// TIA Portal project "Conveyor_Automation_Project" (V17)

(* hardware
DEVICE "S7-1200 station_1"  S7-1200 Station
   slot 0: "Rack_0"  S7-1200 Rack  Rack  V1.0
   slot 1: "PLC_1"  CPU 1214C DC/DC/DC  6ES7 214-1AG40-0XB0  V4.5
DEVICE "HMI_1"  TP700 Comfort
   slot 0: "HMI_1"  TP700 Comfort  6AV2 124-0GC01-0AX0  17.0.0.0
   slot 1: "HMI_RT_1"  TP700 Comfort  6AV2 124-0GC01-0AX0  17.0.0.0
   slot 5: "HMI_1.IE_CP_1"  PROFINET Interface  17.0.0.0
      slot 1: "PROFINET Interface_1"  PROFINET Interface
         slot 1: "Port_1"  Port
         slot 2: "Port_2"  Port
   slot 7: "HMI_1.MPI/DP_CP_1"  MPI/DP Interface  17.0.0.0
*)

// ===== PLC "PLC_1"  CPU 1214C DC/DC/DC =====

VAR_GLOBAL   // PLC tag table "Default tag table"
   "Start_PB" AT %I0.0 : Bool;
   "Stop_PB" AT %I0.1 : Bool;
   "E_Stop" AT %I0.2 : Bool;
   "Object_Sensor" AT %I0.3 : Bool;
   "Sort_Sensor" AT %I0.4 : Bool;
   "Zone1_OL" AT %I0.5 : Bool;
   "Zone2_OL" AT %I0.6 : Bool;
   "Reset_PB" AT %I0.7 : Bool;
   "Zone1_Motor" AT %Q0.0 : Bool;
   "Zone2_Motor" AT %Q0.1 : Bool;
   "Sort_Arm" AT %Q0.2 : Bool;
   "Alarm_Light" AT %Q0.3 : Bool;
   "Run_Light" AT %Q0.4 : Bool;
   "Belt_Speed" AT %IW64 : Word;
   "VFD_Speed_Ref" AT %QW64 : Word;
END_VAR

DATA_BLOCK "Motor1_DB"   // DB1
{ S7_Optimized_Access := 'TRUE' }
VERSION : 0.1
// stored: InstanceOfName Motor_Control
"Motor_Control"
BEGIN
END_DATA_BLOCK

DATA_BLOCK "Safety_DB"   // DB2
{ S7_Optimized_Access := 'TRUE' }
VERSION : 0.1
// stored: InstanceOfName Safety logic
"Safety logic"
BEGIN
END_DATA_BLOCK

DATA_BLOCK "Motor2_DB"   // DB3
{ S7_Optimized_Access := 'TRUE' }
VERSION : 0.1
// stored: InstanceOfName Motor_Control
"Motor_Control"
BEGIN
END_DATA_BLOCK

DATA_BLOCK "Converyor_DB"   // DB4
{ S7_Optimized_Access := 'TRUE' }
VERSION : 0.1
   VAR
      System_RUnning : Bool;
      System_Fault : Bool;
      Safety_Ok : Bool;
      Auto_mode : Bool := true;
      Belt_Speed : Int;
      Belt_Speed_MS : Real;
      VFD_Output : Real;
      Speed_Setpoint : Real := 50.0;
      Good_Count : Int;
      Rject_Count : Int;
      Total_Count : Int;
      Shift_Count : Int;
      Sort_Timer : TON_TIME;
      Jam_timer : TON_TIME;
      Zone2_delay : TON_TIME;
      Good_Count_CTU : CTU_INT;
   END_VAR
   VAR RETAIN
      Reject_Count_CTU : CTU_INT;
      VFD_Output1 : Int;
   END_VAR
   VAR
      Actual_RPM : Real;
   END_VAR
BEGIN
END_DATA_BLOCK

DATA_BLOCK "Alarm_DB"   // DB5
{ S7_Optimized_Access := 'TRUE' }
VERSION : 0.1
   VAR
      Zone1_Fault : Bool;   // Zone 1 motor fault
      Zone2_Fault : Bool;   // Zone 2 motor fault
      E_Stop_Active : Bool;   // E-stop pressed
      Belt_Jam : Bool;   // Belt jam detected
      Speed_Low : Bool;   // Belt speed too low
      Any_Alarm : Bool;   // Any alarm active
      Alarm_Count : Bool;   // Total alarm count
      Alarm_Word : Word;
   END_VAR
BEGIN
END_DATA_BLOCK

DATA_BLOCK "Safety_DB_Instance"   // DB7
{ S7_Optimized_Access := 'TRUE' }
VERSION : 0.1
// stored: InstanceOfName Safety logic
"Safety logic"
BEGIN
END_DATA_BLOCK

DATA_BLOCK "Conveyor_SFC_DB"   // DB8
{ S7_Optimized_Access := 'TRUE' }
VERSION : 0.1
// stored: InstanceOfName Conveyor_SFC
"Conveyor_SFC"
BEGIN
END_DATA_BLOCK

// folder: System blocks/Program resources

DATA_BLOCK "IEC_Timer_0_DB"   // DB6
{ S7_Optimized_Access := 'TRUE' }
AUTHOR : Simatic
FAMILY : IEC
NAME : IEC_TMR
VERSION : 1.0
// stored: InstanceOfName IEC_TIMER
"IEC_TIMER"
BEGIN
END_DATA_BLOCK

// folder: (top level)

FUNCTION_BLOCK "Motor_Control"   // FB1, LAD
{ S7_Optimized_Access := 'TRUE' }
VERSION : 0.1
   VAR_INPUT
      Start : Bool;   // Start command
      Stop : Bool;   // Stop command
      Fault : Bool;   // Motor fault/overload
      Enable : Bool;   // Safety enable signal
      Auto_Mode : Bool;   // Auto or manual mode
   END_VAR
   VAR_OUTPUT
      Motor_Run : Bool;   // Motor output
      Fault_Alarm : Bool;   // Fault active
      Running_FB : Bool;   // Feedback motor running
   END_VAR
   VAR
      Latch : Bool;   // Motor latch memory
      Run_TImer : TON_TIME;   // Confirm run timer
      Fault_Latch : Bool;   // Fault memory
   END_VAR
BEGIN

REGION Network 1: Fault Detection
   // Fault Detection
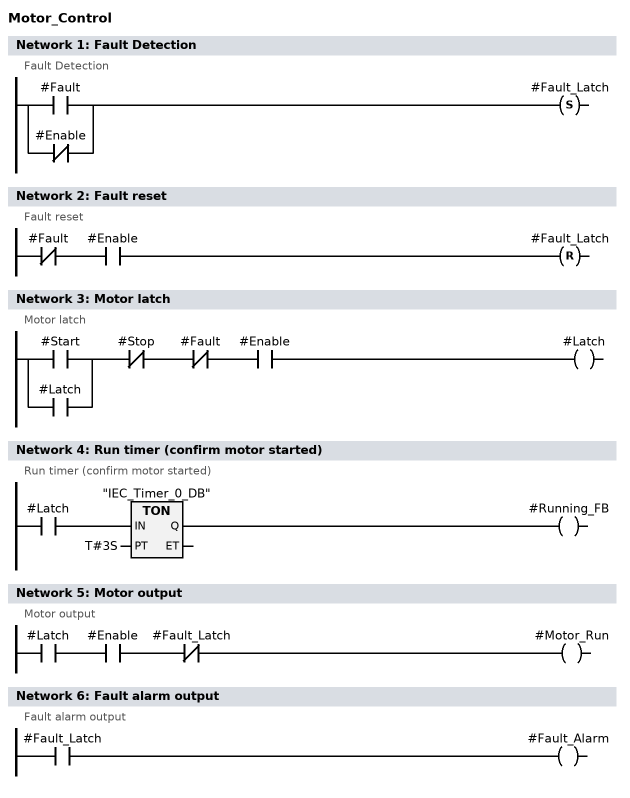
   RUNG wire#powerrail
      Contact( #Fault )
      wire#w1
      S_Coil( #Fault_Latch )
   END_RUNG
   RUNG wire#powerrail
      I_Contact( #Enable )
   END_RUNG wire#w1
   // the same network as SCL:
   IF #Fault OR NOT #Enable THEN #Fault_Latch := TRUE; END_IF;
END_REGION

REGION Network 2: Fault reset
   // Fault reset
   RUNG wire#powerrail
      I_Contact( #Fault )
      Contact( #Enable )
      R_Coil( #Fault_Latch )
   END_RUNG
   // the same network as SCL:
   IF NOT #Fault AND #Enable THEN #Fault_Latch := FALSE; END_IF;
END_REGION

REGION Network 3: Motor latch
   // Motor latch
   RUNG wire#powerrail
      Contact( #Start )
      wire#w1
      I_Contact( #Stop )
      I_Contact( #Fault )
      Contact( #Enable )
      Coil( #Latch )
   END_RUNG
   RUNG wire#powerrail
      Contact( #Latch )
   END_RUNG wire#w1
   // the same network as SCL:
   #Latch := (#Start OR #Latch) AND NOT #Stop AND NOT #Fault AND #Enable;
END_REGION

REGION Network 4: Run timer (confirm motor started)
   // Run timer (confirm motor started)
   "IEC_Timer_0_DB".TON(IN := #Latch, PT := T#3S);
   #Running_FB := "IEC_Timer_0_DB".Q;
END_REGION

REGION Network 5: Motor output
   // Motor output
   RUNG wire#powerrail
      Contact( #Latch )
      Contact( #Enable )
      I_Contact( #Fault_Latch )
      Coil( #Motor_Run )
   END_RUNG
   // the same network as SCL:
   #Motor_Run := #Latch AND #Enable AND NOT #Fault_Latch;
END_REGION

REGION Network 6: Fault alarm output
   // Fault alarm output
   RUNG wire#powerrail
      Contact( #Fault_Latch )
      Coil( #Fault_Alarm )
   END_RUNG
   // the same network as SCL:
   #Fault_Alarm := #Fault_Latch;
END_REGION
END_FUNCTION_BLOCK

FUNCTION_BLOCK "Safety logic"   // FB2, LAD
{ S7_Optimized_Access := 'TRUE' }
VERSION : 0.1
   VAR_INPUT
      E_Stop_Input : Bool;   // E-stop signal (NC — TRUE=OK)
      Gate_Input : Bool;   // Safety gate (NC — TRUE=OK)
      Reset_Input : Bool;   // Reset pushbutton
      Zone1_OL : Bool;   // Zone 1 overload
      Zone2_OL : Bool;   // Zone 2 overload
   END_VAR
   VAR_OUTPUT
      Safety_OK : Bool;   // Safety clear signal
      E_Stop_Active : Bool;   // E-stop alarm
      OL_Active : Bool;   // Overload alarm
   END_VAR
   VAR
      Reset_Latch : Bool;
      Safety_Fault : Bool;
   END_VAR
BEGIN

REGION Network 1: Detect any safety fault
   // Detect any safety fault
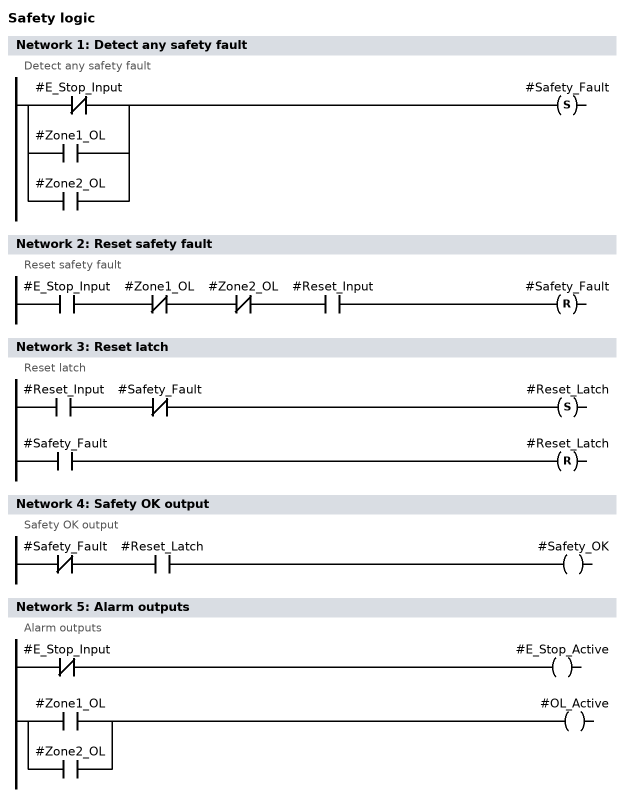
   RUNG wire#powerrail
      I_Contact( #E_Stop_Input )
      wire#w1
      S_Coil( #Safety_Fault )
   END_RUNG
   RUNG wire#powerrail
      Contact( #Zone1_OL )
   END_RUNG wire#w1
   RUNG wire#powerrail
      Contact( #Zone2_OL )
   END_RUNG wire#w1
   // the same network as SCL:
   IF NOT #E_Stop_Input OR #Zone1_OL OR #Zone2_OL THEN #Safety_Fault := TRUE; END_IF;
END_REGION

REGION Network 2: Reset safety fault
   // Reset safety fault
   RUNG wire#powerrail
      Contact( #E_Stop_Input )
      I_Contact( #Zone1_OL )
      I_Contact( #Zone2_OL )
      Contact( #Reset_Input )
      R_Coil( #Safety_Fault )
   END_RUNG
   // the same network as SCL:
   IF #E_Stop_Input AND NOT #Zone1_OL AND NOT #Zone2_OL AND #Reset_Input THEN #Safety_Fault := FALSE; END_IF;
END_REGION

REGION Network 3: Reset latch
   // Reset latch
   RUNG wire#powerrail
      Contact( #Reset_Input )
      I_Contact( #Safety_Fault )
      S_Coil( #Reset_Latch )
   END_RUNG
   RUNG wire#powerrail
      Contact( #Safety_Fault )
      R_Coil( #Reset_Latch )
   END_RUNG
   // the same network as SCL:
   IF #Reset_Input AND NOT #Safety_Fault THEN #Reset_Latch := TRUE; END_IF;
   IF #Safety_Fault THEN #Reset_Latch := FALSE; END_IF;
END_REGION

REGION Network 4: Safety OK output
   // Safety OK output
   RUNG wire#powerrail
      I_Contact( #Safety_Fault )
      Contact( #Reset_Latch )
      Coil( #Safety_OK )
   END_RUNG
   // the same network as SCL:
   #Safety_OK := NOT #Safety_Fault AND #Reset_Latch;
END_REGION

REGION Network 5: Alarm outputs
   // Alarm outputs
   RUNG wire#powerrail
      I_Contact( #E_Stop_Input )
      Coil( #E_Stop_Active )
   END_RUNG
   RUNG wire#powerrail
      Contact( #Zone1_OL )
      wire#w1
      Coil( #OL_Active )
   END_RUNG
   RUNG wire#powerrail
      Contact( #Zone2_OL )
   END_RUNG wire#w1
   // the same network as SCL:
   #E_Stop_Active := NOT #E_Stop_Input;
   #OL_Active := #Zone1_OL OR #Zone2_OL;
END_REGION
END_FUNCTION_BLOCK

FUNCTION_BLOCK "Conveyor_SFC"   // FB3, SCL
{ S7_Optimized_Access := 'TRUE' }
VERSION : 0.1
   VAR_INPUT
      Start_CMD : Bool;   // Start command
      Stop_CMD : Bool;   // Stop command
      Safety_OK : Bool;   // Safety clear
      Zone1_Running : Bool;   // Zone 1 confirmed running
      Object_Detected : Bool;   // Object on belt
      E_Stop : Bool;   // Emergency stop
   END_VAR
   VAR_OUTPUT
      CMD_Zone1_Start : Bool;   // Start Zone1
      CMD_Zone2_Start : Bool;   // Start Zone2
      CMD_Sort : Bool;   // Activate sort arm
      System_State : Int;   // Current state number
   END_VAR
   VAR
      Start_Delay : TON_TIME;
      Stop_Delay : TON_TIME;
   END_VAR
BEGIN
   //====CONVEYOR STATE MACHINE====
   //STATES
   //0 = IDLE
   //1 = STARTING
   //2 = RUNNING
   //3 = SORTING
   //4 = STOPPING
   //5 = STOPPED

   // ----- EMERGENCY STOP FROM ANY STATE -----
   IF NOT #E_Stop OR #Stop_CMD THEN
       #System_State := 4; // JUMP TO STOPPING
   END_IF;

   // --- STATE MACHINE ---
   CASE #System_State OF

       0 :  //IDLE
           #CMD_Zone1_Start := FALSE;
           #CMD_Zone2_Start := FALSE;
           #CMD_Sort := FALSE;
           #Start_Delay(IN := FALSE,
                        PT := T#3S);

           // TRANSITION TO STARTING
           IF #Start_CMD AND #Safety_OK THEN
               #System_State := 1;
           END_IF;

       1 : //STARTING - WAIT 3 SEC
           #CMD_Zone1_Start := FALSE;
           #CMD_Zone2_Start := FALSE;
           #Start_Delay(IN := TRUE,
                        PT := T#3S);

           // TRANSITION TO RUNNING AFTER DELAY
           IF #Start_Delay.Q THEN
               #System_State := 2;
           END_IF;

       2 : //RUNNING - ZONE 1 RUNNING
           #CMD_Zone1_Start := TRUE;
           #CMD_Zone2_Start := FALSE;
           #CMD_Sort := FALSE;
           #Start_Delay(IN := FALSE,
                        PT := T#3S);

           // TRANSITION TO SORTING WHENOBJECT DETECTED
           IF #Object_Detected AND #Zone1_Running THEN
               #System_State := 3;
           END_IF;

       3 : //SORTING - ZONE 2 + SORT ARM ACTIVE
           #CMD_Zone1_Start := TRUE;
           #CMD_Zone2_Start := TRUE;
           #CMD_Sort := TRUE;

           // TRANSITION BACK TO RUNNING WHEN OBJECT PASSED
           IF NOT #Object_Detected THEN
               #System_State := 2;
           END_IF;

       4 : //STOPPING - RAMP DOWN
           #CMD_Zone1_Start := FALSE;
           #CMD_Zone2_Start := FALSE;
           #CMD_Sort := FALSE;
           #Stop_Delay(IN := TRUE,
                       PT := T#2S);

           // TRANSITION TO STOPPED
           IF #Stop_Delay.Q THEN
               #System_State := 5;
           END_IF;

       5 :
           #Stop_Delay(IN := FALSE,
                       PT := T#2S);
           #System_State := 0; // AUTO BACK TO IDLE

       ELSE  // Statement section ELSE
           #System_State := 0; // SAFETY - UNKNOWN STATE

   END_CASE;
END_FUNCTION_BLOCK

FUNCTION "Analog Scaling" : Void   // FC1, SCL
{ S7_Optimized_Access := 'TRUE' }
VERSION : 0.1
   VAR_INPUT
      Raw_Value : Int;
      Eng_Min : Real;
      Eng_Max : Real;
      Raw_Min : Int;
      Raw_Max : Int;
   END_VAR
   VAR_OUTPUT
      Eng_Value : Real;
   END_VAR
BEGIN
   // Wire break detection
   IF #Raw_Value < 1000 THEN
       #Eng_Value := 0.0;
       RETURN;
   END_IF;

   // Overflow detection  
   IF #Raw_Value > 28000 THEN
       #Eng_Value := #Eng_Max;
       RETURN;
   END_IF;


   #Eng_Value := (INT_TO_REAL(#Raw_Value - #Raw_Min) *
   (#Eng_Max - #Eng_Min)) /
   INT_TO_REAL(#Raw_Max - #Raw_Min) +
   #Eng_Min;
END_FUNCTION

FUNCTION "Alarm Handler" : Void   // FC2, SCL
{ S7_Optimized_Access := 'TRUE' }
VERSION : 0.1
BEGIN
END_FUNCTION

FUNCTION "Counter Logic" : Void   // FC3, LAD
{ S7_Optimized_Access := 'TRUE' }
VERSION : 0.1
BEGIN
END_FUNCTION

ORGANIZATION_BLOCK "Main"   // OB1, SCL, ProgramCycle
TITLE = "Main Program Sweep (Cycle)"
{ S7_Optimized_Access := 'TRUE' }
VERSION : 0.1
   VAR_INPUT
      Initial_Call : Bool;   // Initial call of this OB
      Remanence : Bool;   // =True, if remanent data are available
   END_VAR
BEGIN
   // ═══════════════════════════════════════
   // CONVEYOR AUTOMATION — MAIN PROGRAM
   // Author: Ujwala Venuturla
   // Date: 2026
   // ═══════════════════════════════════════

   // ---SFC SEQUENCE CONTROLLER ---
   "Conveyor_SFC_DB"(Start_CMD := "Start_PB",
                     Stop_CMD := "Stop_PB",
                     Safety_OK := "Converyor_DB".Safety_Ok,
                     Zone1_Running := "Motor1_DB".Running_FB,
                     Object_Detected := "Object_Sensor",
                     E_Stop := NOT "E_Stop");

   //----STEP 1: SAFETY LOGIC ------
   "Safety_DB_Instance"(
                      E_Stop_Input := "E_Stop",
                      Gate_Input   := TRUE,
                      Reset_Input  := "Reset_PB",
                      Zone1_OL := "Zone1_OL",
                      Zone2_OL := "Zone2_OL");

   //Store Safety Status
   "Converyor_DB".Safety_Ok := "Safety_DB_Instance".Safety_OK;

   //-----STEP 2 : ZONE1 MOTOR----
   "Motor1_DB"(
               Start := "Start_PB" AND "Converyor_DB".Safety_Ok,
               Stop  := "Stop_PB",
               Fault := "Zone1_OL",
               Enable := "Converyor_DB".Safety_Ok,
               Auto_Mode := TRUE);
   "Zone1_Motor" := "Motor1_DB".Motor_Run;
   "Run_Light" := "Motor1_DB".Motor_Run;

   //-----STEP3:ZONE 2 MOTOR----
   //ZONE 2 STARTS ONLY WHEN OBJECT DETECTED AND ZONE 1 IS RUNNING
   "Motor2_DB"(
               Start := "Object_Sensor" AND "Motor1_DB".Motor_Run,
               Stop  := "Stop_PB",
               Fault := "Zone2_OL",
               Enable := "Converyor_DB".Safety_Ok,
               Auto_Mode := TRUE);

   "Zone2_Motor" := "Motor2_DB".Motor_Run;

   //----STEP 4: SORTING ARM LOGIC----
   //SORTING ARM ACTIVATES WHEN SORT SENSOR TRUE AND ZONE2 MOTOR RUNNING
   "Converyor_DB".Sort_Timer(
                             IN := "Sort_Sensor" AND "Motor2_DB".Motor_Run,
                             PT := T#2S);

   "Sort_Arm" := "Converyor_DB".Sort_Timer.Q;

   //STEP 5 : COUNTER LOGIC
   //COUNTS GOOD OBJECTS (SORT SENSOR FALSE = GOOD)
   "Converyor_DB".Good_Count_CTU(CU := "Object_Sensor" AND NOT "Sort_Sensor",
                             R:="Reset_PB",
                             PV := 9999);

   //// Count rejected objects (sort sensor TRUE = reject)
   "Converyor_DB".Reject_Count_CTU(CU := "Object_Sensor" AND "Sort_Sensor",
                                   R  := "Reset_PB",
                                   PV := 9999);

   // Total count
   "Converyor_DB".Total_Count := "Converyor_DB".Good_Count_CTU.CV + "Converyor_DB".Reject_Count_CTU.CV;

   //-----STEP 6 : Analog Speed Scaling---
   "Analog Scaling"(
                    Raw_Value := "Belt_Speed",
                    Eng_Min := 0.0,
                    Eng_Max := 3.0,
                    Raw_Min := 0,
                    Raw_Max := 27648,
                    Eng_Value => "Converyor_DB".Belt_Speed_MS);

   //----STEP 7: ALARM LOGIC
   "Converyor_DB".System_Fault := "Motor1_DB".Fault_Alarm
   OR "Motor2_DB".Fault_Alarm
   OR "Safety_DB_Instance".E_Stop_Active;

   "Alarm_Light" := "Converyor_DB".System_Fault;

   //----STEP 8 : SYSTEM RUNNING STATUS
   "Converyor_DB".System_RUnning := "Motor1_DB".Motor_Run;

   // Pack alarms into Alarm_Word
   "Alarm_DB".Alarm_Word.%X0 := "Motor1_DB".Fault_Alarm;
   "Alarm_DB".Alarm_Word.%X1 := "Motor2_DB".Fault_Alarm;
   "Alarm_DB".Alarm_Word.%X2 := "Safety_DB_Instance".E_Stop_Active;
   "Alarm_DB".Alarm_Word.%X3 := "Zone1_OL";
   "Alarm_DB".Alarm_Word.%X4 := "Zone2_OL";

   //---VFD SPEED CONTROL ---
   //// Convert speed setpoint (0-100%) to analog output (0-27648)
   IF "Converyor_DB".System_RUnning THEN
       "Converyor_DB".VFD_Output1 := REAL_TO_INT("Converyor_DB".Speed_Setpoint / 100 *27648.0);
   ELSE
       "Converyor_DB".VFD_Output := 0;
   END_IF;

   //---Write to analog output---
   "VFD_Speed_Ref" := "Converyor_DB".VFD_Output1 ;

   //Read actual belt speed back
   "Analog Scaling"(
                    Raw_Value := "Belt_Speed",
                    Eng_Min := 0.0,
                    Eng_Max := 1500.0,
                    Raw_Min := 0,
                    Raw_Max := 27648,
                    Eng_Value => "Converyor_DB".Actual_RPM);
END_ORGANIZATION_BLOCK

(* ===== HMI "HMI_RT_1" =====
system functions are stored by id; their names below are inferred from use
connection "HMI_Connection_1": ETHERNET, S7_1200_OMS

HMI tags "Default tag table"
   "Tag_ScreenNumber" : UInt, internal
   "Zone1_Status" : Bool = PLC Motor1_DB.Motor_Run, 1 s
   "Zone2_Status" : Bool = PLC Motor2_DB.Motor_Run, 1 s
   "Sort_Status" : Bool = PLC Sort_Arm AT %Q0.2, 1 s
   "Good_Count" : Int = PLC Converyor_DB.Good_Count_CTU.CV AT %DB1.DBX0.0, 1 s
   "Reject_Count" : Int = PLC Converyor_DB.Reject_Count_CTU.CV AT %DB1.DBX0.0, 1 s
   "Total_Count" : Int = PLC Converyor_DB.Total_Count AT %DB1.DBX0.0, 1 s
   "System_Fault" : Bool = PLC Converyor_DB.System_Fault AT %DB1.DBW0, 1 s
   "Belt_Speed" : Real = PLC Converyor_DB.Belt_Speed_MS AT %DB1.DBW0, 1 s
   "System_State" : Int = PLC Conveyor_SFC_DB.System_State AT %DB1.DBW0, 1 s
   "Safety_Status" : Bool = PLC Converyor_DB.Safety_Ok AT %DB1.DBW0, 1 s
   "Start_PB" : Bool = PLC Start_PB AT %I0.0, 1 s
   "Stop_PB" : Bool = PLC Stop_PB AT %I0.1, 1 s
   "Reset_PB" : Bool = PLC Reset_PB AT %I0.7, 1 s
   "Motor1_Fault" : Bool = PLC Motor1_DB.Fault_Alarm AT %DB1.DBX0.0, 1 s
   "Motor2_Fault" : Bool = PLC Motor2_DB.Fault_Alarm AT %DB1.DBX0.0, 1 s
   "Emergency Stop" : Bool = PLC Safety_DB_Instance.E_Stop_Active AT %DB1.DBX0.0, 1 s
   "Zone1 Overload" : Bool = PLC Safety_DB_Instance.Zone1_OL AT %DB1.DBX0.0, 1 s
   "Zone2 Overload" : Bool = PLC Safety_DB_Instance.Zone2_OL AT %DB1.DBX0.0, 1 s
   "Alarm_Word" : Word = PLC Alarm_DB.Alarm_Word AT %DB1.DBW0, 1 s
   "Converyor_DB_Speed_Setpoint" : Real = PLC Converyor_DB.Speed_Setpoint, 1 s
   "Converyor_DB_Actual_RPM" : Real = PLC Converyor_DB.Actual_RPM, 1 s

HMI tags "Tag table_1"
   "HMI_Tag_1" : Int, internal

discrete alarms
   1: 'Zone 1 Motor Fault', class Errors, trigger "Alarm_Word" bit 0
   2: 'Zone 2 Motor Fault', class Errors, trigger "Alarm_Word" bit 1
   3: 'Emergency Stop', class Errors, trigger "Alarm_Word" bit 2
   4: 'Zone 1 Overload', class Warnings, trigger "Alarm_Word" bit 3
   5: 'Zone 2 Overload', class Warnings, trigger "Alarm_Word" bit 4

text list "System_Status": 0 'IDLE'; 1 'STARTING'; 2 'RUNNING'; 3 'SORTING'; 4 'STOPPING'

screen "Home_Screen" 800x420, template "Template_1"
   on GenerateScreen: SetTag("Tag_ScreenNumber", 1)
   Button "Button_1" at 87,40 size 75x32; TextOff 'START'
      on Click: SetBit("Start_PB")
   Button "Button_2" at 168,40 size 75x32; TextOff 'STOP'
      on Click: SetBit("Stop_PB")
   Button "Button_3" at 248,40 size 75x32; TextOff 'RESET'
      on Click: SetBit("Stop_PB")
   Circle "Circle_1" at 87,113 size 27x27
      Appearance <- "Zone1_Status"
   Circle "Circle_2" at 212,113 size 27x27
      Appearance <- "Zone2_Status"
   Circle "Circle_3" at 349,113 size 27x27
      Appearance <- "Sort_Status"
   TextField "Text field_1" at 123,114 size 88x26; Text 'ZONE 1'
   TextField "Text field_2" at 244,114 size 82x26; Text 'ZONE 2'
   TextField "Text field_3" at 380,115 size 101x26; Text 'SORT ARM'
   TextField "Text field_4" at 390,43 size 69x26; Text 'STATE :'
   TextField "Text field_5" at 87,170 size 76x26; Text 'GOOD :'
   SymbolicIOField "Symbolic I/O field_1" at 509,40 size 65x32; TextOff '0'; TextOn '1'; TextList "System_Status"
      ProcessValue <- "System_State"
   IOField "I/O field_1" at 462,40 size 36x32; FormatPattern 9
      ProcessValue <- "System_State"
   IOField "I/O field_2" at 163,167 size 54x32; FormatPattern 999
      ProcessValue <- "Good_Count"
   TextField "Text field_6" at 248,170 size 80x26; Text 'REJECT :'
   TextField "Text field_7" at 418,167 size 69x26; Text 'TOTAL :'
   IOField "I/O field_3" at 326,167 size 54x32; FormatPattern 999
      ProcessValue <- "Good_Count"
   IOField "I/O field_4" at 487,167 size 54x32; FormatPattern 999
      ProcessValue <- "Good_Count"
   TextField "Text field_8" at 87,218 size 118x26; Text 'BELT SPEED :'
   TextField "Text field_9" at 87,266 size 161x26; Text '⚠ SYSTEM FAULT'
      Visibility <- "System_Fault"
   Button "Button_4" at 640,362 size 75x57; TextOff 'ALARMS'
      on Click: ActivateScreen("Alarm_Screen", 0)
   Button "Button_5" at 561,362 size 75x57; TextOff 'TRENDS'
      on Click: ActivateScreen("Trend_Screen", 0)
   Button "Button_6" at 480,362 size 77x57; TextOff 'COUNTER'
      on Click: ActivateScreen("Counter_Screen", 0)
   Bar "Bar_1" at 205,218 size 172x35; MinimumValue 0; MaximumValue 3
      ProcessValue <- "Belt_Speed"
   IOField "I/O field_5" at 619,78 size 96x32; FormatPattern 999
      ProcessValue <- "Converyor_DB_Speed_Setpoint"
   TextField "Text field_10" at 531,82 size 87x26; Text 'Speed SP :'
   IOField "I/O field_6" at 619,126 size 96x32; FormatPattern 999
      ProcessValue <- "Converyor_DB_Actual_RPM"
   TextField "Text field_11" at 531,130 size 87x26; Text 'Actual RPM:'

Template "Template_1" 800x420
   Button "Exit" at 720,360 size 78x58; TextOff 'Exit'; PictureOff "ExitRuntime_TP700_Comfort_TR"; PictureOn "ExitRuntime_TP700_Comfort_TR"
      on Release: StopRuntime(0)
   Button "Template_Button" at 640,360 size 78x58; TextOff 'Text'
   Button "Template_Button_1" at 560,360 size 78x58; TextOff 'Text'
   Button "Template_Button_2" at 480,360 size 78x58; TextOff 'Text'
   Button "Template_Button_3" at 400,360 size 78x58; TextOff 'Text'
   Button "Template_Button_4" at 321,360 size 78x58; TextOff 'Text'
   Button "Template_Button_5" at 241,360 size 78x58; TextOff 'Text'
   Button "Template_Button_6" at 161,360 size 78x58; TextOff 'Text'
   Button "Alarms" at 81,360 size 78x58; TextOff 'Alarms'; PictureOff "AlarmDisplay_TP700_Comfort_TR"; PictureOn "AlarmDisplay_TP700_Comfort_TR"
      on Release: function_ef3f5d25("Alarm window_Unacknowledged", -1)
   Button "Start screen" at 1,360 size 78x58; TextOff 'Start screen'; PictureOff "NavigateHome_TP700_Comfort_TR"; PictureOn "NavigateHome_TP700_Comfort_TR"
      on Release: ActivateScreen("Home_Screen", 0)

screen "Trend_Screen" 800x420
   TrendView "Trend view_1" at 11,12 size 658x356
   Button "Button_1" at 719,359 size 58x50; TextOff 'BACK'
      on Click: ActivateScreen("Home_Screen", 0)

screen "Counter_Screen" 800x420
   IOField "I/O field_1" at 329,47 size 96x32; FormatPattern 999
      ProcessValue <- "Good_Count"
   IOField "I/O field_2" at 329,111 size 96x32; FormatPattern 999
      ProcessValue <- "Reject_Count"
   IOField "I/O field_3" at 329,175 size 96x32; FormatPattern 999
      ProcessValue <- "Total_Count"
   TextField "Text field_1" at 186,49 size 112x23; Text 'Good Parts:'
   TextField "Text field_2" at 186,115 size 147x23; Text 'Rejected Parts:'
   TextField "Text field_3" at 186,181 size 119x23; Text 'Total Count:'
   Button "Button_1" at 615,50 size 96x32; TextOff 'RESET'
      on Click: SetBit("Reset_PB")
   TextField "Text field_4" at 600,88 size 135x23; Text 'Counter Reset'
   Button "Button_2" at 719,359 size 58x50; TextOff 'BACK'
      on Click: ActivateScreen("Home_Screen", 0)
*)